(* PLC project Adressering.ecp, WAGO e!COCKPIT e!COCKPIT *)
(* stored: creationDateTime 2021-01-18T14:20:23.2110188, modificationDateTime 2021-01-18T11:51:27.6823754 *)

TYPE dtRomtype_1 : STRUCT
  RB601_V : BOOL;  (* Bevegelse *)
END_STRUCT;
END_TYPE

TYPE dtRomtype_11 : STRUCT
  RB601_V : BOOL;  (* Bevegelse *)
  RB601_HVAC : BOOL;  (* HVAC signal *)
END_STRUCT;
END_TYPE

TYPE dtRomtype_111 : STRUCT
  RB601_V : BOOL;  (* Bevegelse *)
  RB601_HVAC : BOOL;  (* HVAC signal *)
  RT601_CT : REAL;  (* Rom temperatur *)
  RT601_SP_D : REAL;  (* Temperatur SP dag/komfort *)
  RT601_SP_S : REAL;  (* Temperatur SP standby *)
  RT601_SP_N : REAL;  (* Temperatur SP nattsenk *)
  RT601_SP_F : REAL;  (* Temperatur SP frostsikring *)
  RT601_CS : REAL;  (* Aktivt temperatur SP *)
  OPM : REAL;  (* Rom modus *)
  OPM_CV : REAL;  (* Rom modus verdi *)
END_STRUCT;
END_TYPE

TYPE dtRomtype_1111 : STRUCT
  RB601_V : BOOL;  (* Bevegelse *)
  RB601_HVAC : BOOL;  (* HVAC signal *)
  RT601_CT : REAL;  (* Rom temperatur *)
  RT601_SP_D : REAL;  (* Temperatur SP dag/komfort *)
  RT601_SP_S : REAL;  (* Temperatur SP standby *)
  RT601_SP_N : REAL;  (* Temperatur SP nattsenk *)
  RT601_SP_F : REAL;  (* Temperatur SP frostsikring *)
  RT601_CS : REAL;  (* Aktivt temperatur SP *)
  OPM : REAL;  (* Rom modus *)
  OPM_CV : REAL;  (* Rom modus verdi *)
  RY601_CV : REAL;  (* Co2 Nivaa *)
  RY601_SP : REAL;  (* Co2 SP *)
  RY601_OP : REAL;  (* Co2 paadrag *)
END_STRUCT;
END_TYPE

TYPE dtRomtype_11101 : STRUCT
  RB601_V : BOOL;  (* Bevegelse *)
  RB601_HVAC : BOOL;  (* HVAC signal *)
  RT601_CT : REAL;  (* Rom temperatur *)
  RT601_SP_D : REAL;  (* Temperatur SP dag/komfort *)
  RT601_SP_S : REAL;  (* Temperatur SP standby *)
  RT601_SP_N : REAL;  (* Temperatur SP nattsenk *)
  RT601_SP_F : REAL;  (* Temperatur SP frostsikring *)
  RT601_CS : REAL;  (* Aktivt temperatur SP *)
  OPM : REAL;  (* Rom modus *)
  OPM_CV : REAL;  (* Rom modus verdi *)
  LH601_OP : REAL;  (* Varmepaadrag *)
  SB601_MAN : REAL;  (* Varmepaadrag force *)
END_STRUCT;
END_TYPE

TYPE dtRomtype_111011 : STRUCT
  RB601_V : BOOL;  (* Bevegelse *)
  RB601_HVAC : BOOL;  (* HVAC signal *)
  RT601_CT : REAL;  (* Rom temperatur *)
  RT601_SP_D : REAL;  (* Temperatur SP dag/komfort *)
  RT601_SP_S : REAL;  (* Temperatur SP standby *)
  RT601_SP_N : REAL;  (* Temperatur SP nattsenk *)
  RT601_SP_F : REAL;  (* Temperatur SP frostsikring *)
  RT601_CS : REAL;  (* Aktivt temperatur SP *)
  OPM : REAL;  (* Rom modus *)
  OPM_CV : REAL;  (* Rom modus verdi *)
  LH601_OP : REAL;  (* Varmepaadrag *)
  SB601_MAN : REAL;  (* Varmepaadrag force *)
  LH601_CMD : BOOL;  (* LH601_CMD *)
END_STRUCT;
END_TYPE

TYPE dtRomtype_1110111 : STRUCT
  RB601_V : BOOL;  (* Bevegelse *)
  RB601_HVAC : BOOL;  (* HVAC signal *)
  RT601_CT : REAL;  (* Rom temperatur *)
  RT601_SP_D : REAL;  (* Temperatur SP dag/komfort *)
  RT601_SP_S : REAL;  (* Temperatur SP standby *)
  RT601_SP_N : REAL;  (* Temperatur SP nattsenk *)
  RT601_SP_F : REAL;  (* Temperatur SP frostsikring *)
  RT601_CS : REAL;  (* Aktivt temperatur SP *)
  OPM : REAL;  (* Rom modus *)
  OPM_CV : REAL;  (* Rom modus verdi *)
  LH601_OP : REAL;  (* Varmepaadrag *)
  SB601_MAN : REAL;  (* Varmepaadrag force *)
  LH601_CMD : BOOL;  (* LH601_CMD *)
  LC601_OP : REAL;  (* LC601_OP *)
  LC601_MAN : REAL;  (* LC601 Force *)
END_STRUCT;
END_TYPE

TYPE dtRomtype_11111111 : STRUCT
  RB601_V : BOOL;  (* Bevegelse *)
  RB601_HVAC : BOOL;  (* HVAC signal *)
  RT601_CT : REAL;  (* Rom temperatur *)
  RT601_SP_D : REAL;  (* Temperatur SP dag/komfort *)
  RT601_SP_S : REAL;  (* Temperatur SP standby *)
  RT601_SP_N : REAL;  (* Temperatur SP nattsenk *)
  RT601_SP_F : REAL;  (* Temperatur SP frostsikring *)
  RT601_CS : REAL;  (* Aktivt temperatur SP *)
  OPM : REAL;  (* Rom modus *)
  OPM_CV : REAL;  (* Rom modus verdi *)
  RY601_CV : REAL;  (* Co2 Nivaa *)
  RY601_SP : REAL;  (* Co2 SP *)
  RY601_OP : REAL;  (* Co2 paadrag *)
  LH601_OP : REAL;  (* Varmepaadrag *)
  SB601_MAN : REAL;  (* Varmepaadrag force *)
  LH601_CMD : BOOL;  (* LH601_CMD *)
  LC601_OP : REAL;  (* LC601_OP *)
  LC601_MAN : REAL;  (* LC601 Force *)
  LC601_CMD : BOOL;  (* LC601_CMD *)
END_STRUCT;
END_TYPE

TYPE dtRomtype_111010111 : STRUCT
  RB601_V : BOOL;  (* Bevegelse *)
  RB601_HVAC : BOOL;  (* HVAC signal *)
  RT601_CT : REAL;  (* Rom temperatur *)
  RT601_SP_D : REAL;  (* Temperatur SP dag/komfort *)
  RT601_SP_S : REAL;  (* Temperatur SP standby *)
  RT601_SP_N : REAL;  (* Temperatur SP nattsenk *)
  RT601_SP_F : REAL;  (* Temperatur SP frostsikring *)
  RT601_CS : REAL;  (* Aktivt temperatur SP *)
  OPM : REAL;  (* Rom modus *)
  OPM_CV : REAL;  (* Rom modus verdi *)
  LH601_OP : REAL;  (* Varmepaadrag *)
  SB601_MAN : REAL;  (* Varmepaadrag force *)
  LC601_OP : REAL;  (* LC601_OP *)
  LC601_MAN : REAL;  (* LC601 Force *)
  LC601_CMD : BOOL;  (* LC601_CMD *)
  RT601_SP : REAL;  (* Temperatur SP feedback *)
END_STRUCT;
END_TYPE

TYPE dtRomtype_1111101011 : STRUCT
  RB601_V : BOOL;  (* Bevegelse *)
  RB601_HVAC : BOOL;  (* HVAC signal *)
  RT601_CT : REAL;  (* Rom temperatur *)
  RT601_SP_D : REAL;  (* Temperatur SP dag/komfort *)
  RT601_SP_S : REAL;  (* Temperatur SP standby *)
  RT601_SP_N : REAL;  (* Temperatur SP nattsenk *)
  RT601_SP_F : REAL;  (* Temperatur SP frostsikring *)
  RT601_CS : REAL;  (* Aktivt temperatur SP *)
  OPM : REAL;  (* Rom modus *)
  OPM_CV : REAL;  (* Rom modus verdi *)
  RY601_CV : REAL;  (* Co2 Nivaa *)
  RY601_SP : REAL;  (* Co2 SP *)
  RY601_OP : REAL;  (* Co2 paadrag *)
  LH601_OP : REAL;  (* Varmepaadrag *)
  SB601_MAN : REAL;  (* Varmepaadrag force *)
  LC601_OP : REAL;  (* LC601_OP *)
  LC601_MAN : REAL;  (* LC601 Force *)
  RT601_SP : REAL;  (* Temperatur SP feedback *)
  RT601_SP_FB : REAL;  (* Temperatur SP *)
  RT601_SP_IN : REAL;  (* Temperatur SP lokalt panel *)
END_STRUCT;
END_TYPE

TYPE dtRomtype_1111111111 : STRUCT
  RB601_V : BOOL;  (* Bevegelse *)
  RB601_HVAC : BOOL;  (* HVAC signal *)
  RT601_CT : REAL;  (* Rom temperatur *)
  RT601_SP_D : REAL;  (* Temperatur SP dag/komfort *)
  RT601_SP_S : REAL;  (* Temperatur SP standby *)
  RT601_SP_N : REAL;  (* Temperatur SP nattsenk *)
  RT601_SP_F : REAL;  (* Temperatur SP frostsikring *)
  RT601_CS : REAL;  (* Aktivt temperatur SP *)
  OPM : REAL;  (* Rom modus *)
  OPM_CV : REAL;  (* Rom modus verdi *)
  RY601_CV : REAL;  (* Co2 Nivaa *)
  RY601_SP : REAL;  (* Co2 SP *)
  RY601_OP : REAL;  (* Co2 paadrag *)
  LH601_OP : REAL;  (* Varmepaadrag *)
  SB601_MAN : REAL;  (* Varmepaadrag force *)
  LH601_CMD : BOOL;  (* LH601_CMD *)
  LC601_OP : REAL;  (* LC601_OP *)
  LC601_MAN : REAL;  (* LC601 Force *)
  LC601_CMD : BOOL;  (* LC601_CMD *)
  RT601_SP : REAL;  (* Temperatur SP feedback *)
  RT601_SP_FB : REAL;  (* Temperatur SP *)
  RT601_SP_IN : REAL;  (* Temperatur SP lokalt panel *)
END_STRUCT;
END_TYPE

{attribute 'qualified_only'}
VAR_GLOBAL  (* STLV80_563 *)
  STLV80_A_563_KNX_Card_1_Status : BOOL;  (* KNX kort 1 status *)
  STLV80_A_563_5A201 : dtRomtype_1;  (* rom1 *)
  STLV80_A_563_5A202 : dtRomtype_11;  (* rom1 *)
  STLV80_A_563_5A301 : dtRomtype_111;  (* rom1 *)
  STLV80_A_563_5A302 : dtRomtype_1111;  (* rom1 *)
  STLV80_A_563_5B201 : dtRomtype_11101;  (* rom1 *)
  STLV80_A_563_5B202 : dtRomtype_111011;  (* rom1 *)
  STLV80_A_563_5B301 : dtRomtype_1110111;  (* rom1 *)
  STLV80_A_563_5B302 : dtRomtype_11111111;  (* rom1 *)
  STLV80_A_563_5C201 : dtRomtype_111010111;  (* rom1 *)
  STLV80_A_563_5C202 : dtRomtype_1111101011;  (* rom1 *)
  STLV80_A_563_5C301 : dtRomtype_11111111;  (* rom1 *)
  STLV80_A_563_5C302 : dtRomtype_1111111111;  (* rom1 *)
  STLV80_A_563_5D201 : dtRomtype_1111111111;  (* rom1 *)
  STLV80_A_563_5D202 : dtRomtype_1111111111;  (* rom1 *)
  STLV80_A_563_5D301 : dtRomtype_1111111111;  (* rom1 *)
  STLV80_A_563_5D302 : dtRomtype_1111111111;  (* rom1 *)
END_VAR

PROGRAM PRG_563_KNX_1
  VAR
    i : INT := 0;  (* Felles *)
    Interval : OSCAT_BASIC.CLK_PRG;
    typDPT : typDPT;
    KNX_master_1 : WagoAppKNX.FbKNX_Master;  (* Master *)
    M1_001_5A201_RB601_V : fbDPT_Switch_pro;  (* 5A201 *)
    M1_002_5A202_RB601_V : fbDPT_Switch_pro;  (* 5A202 *)
    M1_003_5A202_RB601_HVAC : fbDPT_Switch_pro;  (* 5A202 *)
    M1_004_5A301_RB601_V : fbDPT_Switch_pro;  (* 5A301 *)
    M1_005_5A301_RB601_HVAC : fbDPT_Switch_pro;  (* 5A301 *)
    M1_006_5A301_RT601_CT : fbDPT_Value_Temp_pro;  (* 5A301 *)
    M1_007_5A302_RB601_V : fbDPT_Switch_pro;  (* 5A302 *)
    M1_008_5A302_RB601_HVAC : fbDPT_Switch_pro;  (* 5A302 *)
    M1_009_5A302_RT601_CT : fbDPT_Value_Temp_pro;  (* 5A302 *)
    M1_010_5A302_RY601_CV : fbDPT_Value_AirQuality_pro;  (* 5A302 *)
    M1_011_5B201_RB601_V : fbDPT_Switch_pro;  (* 5B201 *)
    M1_012_5B201_RB601_HVAC : fbDPT_Switch_pro;  (* 5B201 *)
    M1_013_5B201_RT601_CT : fbDPT_Value_Temp_pro;  (* 5B201 *)
    M1_014_5B201_LH601_OP : fbDPT_Scaling_pro;  (* 5B201 *)
    M1_015_5B202_RB601_V : fbDPT_Switch_pro;  (* 5B202 *)
    M1_016_5B202_RB601_HVAC : fbDPT_Switch_pro;  (* 5B202 *)
    M1_017_5B202_RT601_CT : fbDPT_Value_Temp_pro;  (* 5B202 *)
    M1_018_5B202_LH601_OP : fbDPT_Scaling_pro;  (* 5B202 *)
    M1_019_5B202_LH601_CMD : fbDPT_Switch_pro;  (* 5B202 *)
    M1_020_5B301_RB601_V : fbDPT_Switch_pro;  (* 5B301 *)
    M1_021_5B301_RB601_HVAC : fbDPT_Switch_pro;  (* 5B301 *)
    M1_022_5B301_RT601_CT : fbDPT_Value_Temp_pro;  (* 5B301 *)
    M1_023_5B301_LH601_OP : fbDPT_Scaling_pro;  (* 5B301 *)
    M1_024_5B301_LH601_CMD : fbDPT_Switch_pro;  (* 5B301 *)
    M1_025_5B301_LC601_OP : fbDPT_Scaling_pro;  (* 5B301 *)
    M1_026_5B302_RB601_V : fbDPT_Switch_pro;  (* 5B302 *)
    M1_027_5B302_RB601_HVAC : fbDPT_Switch_pro;  (* 5B302 *)
    M1_028_5B302_RT601_CT : fbDPT_Value_Temp_pro;  (* 5B302 *)
    M1_029_5B302_RY601_CV : fbDPT_Value_AirQuality_pro;  (* 5B302 *)
    M1_030_5B302_LH601_OP : fbDPT_Scaling_pro;  (* 5B302 *)
    M1_031_5B302_LH601_CMD : fbDPT_Switch_pro;  (* 5B302 *)
    M1_032_5B302_LC601_OP : fbDPT_Scaling_pro;  (* 5B302 *)
    M1_033_5B302_LC601_CMD : fbDPT_Switch_pro;  (* 5B302 *)
    M1_034_5C201_RB601_V : fbDPT_Switch_pro;  (* 5C201 *)
    M1_035_5C201_RB601_HVAC : fbDPT_Switch_pro;  (* 5C201 *)
    M1_036_5C201_RT601_CT : fbDPT_Value_Temp_pro;  (* 5C201 *)
    M1_037_5C201_LH601_OP : fbDPT_Scaling_pro;  (* 5C201 *)
    M1_038_5C201_LC601_OP : fbDPT_Scaling_pro;  (* 5C201 *)
    M1_039_5C201_LC601_CMD : fbDPT_Switch_pro;  (* 5C201 *)
    M1_040_5C201_RT601_SP : fbDPT_Value_Temp_pro;  (* 5C201 *)
    M1_041_5C202_RB601_V : fbDPT_Switch_pro;  (* 5C202 *)
    M1_042_5C202_RB601_HVAC : fbDPT_Switch_pro;  (* 5C202 *)
    M1_043_5C202_RT601_CT : fbDPT_Value_Temp_pro;  (* 5C202 *)
    M1_044_5C202_RY601_CV : fbDPT_Value_AirQuality_pro;  (* 5C202 *)
    M1_045_5C202_LH601_OP : fbDPT_Scaling_pro;  (* 5C202 *)
    M1_046_5C202_LC601_OP : fbDPT_Scaling_pro;  (* 5C202 *)
    M1_047_5C202_RT601_SP : fbDPT_Value_Temp_pro;  (* 5C202 *)
    M1_048_5C202_RT601_SP_FB : fbDPT_Value_Temp_pro;  (* 5C202 *)
    M1_049_5C301_RB601_V : fbDPT_Switch_pro;  (* 5C301 *)
    M1_050_5C301_RB601_HVAC : fbDPT_Switch_pro;  (* 5C301 *)
    M1_051_5C301_RT601_CT : fbDPT_Value_Temp_pro;  (* 5C301 *)
    M1_052_5C301_RY601_CV : fbDPT_Value_AirQuality_pro;  (* 5C301 *)
    M1_053_5C301_LH601_OP : fbDPT_Scaling_pro;  (* 5C301 *)
    M1_054_5C301_LH601_CMD : fbDPT_Switch_pro;  (* 5C301 *)
    M1_055_5C301_LC601_OP : fbDPT_Scaling_pro;  (* 5C301 *)
    M1_056_5C301_LC601_CMD : fbDPT_Switch_pro;  (* 5C301 *)
    M1_057_5C302_RB601_V : fbDPT_Switch_pro;  (* 5C302 *)
    M1_058_5C302_RB601_HVAC : fbDPT_Switch_pro;  (* 5C302 *)
    M1_059_5C302_RT601_CT : fbDPT_Value_Temp_pro;  (* 5C302 *)
    M1_060_5C302_RY601_CV : fbDPT_Value_AirQuality_pro;  (* 5C302 *)
    M1_061_5C302_LH601_OP : fbDPT_Scaling_pro;  (* 5C302 *)
    M1_062_5C302_LH601_CMD : fbDPT_Switch_pro;  (* 5C302 *)
    M1_063_5C302_LC601_OP : fbDPT_Scaling_pro;  (* 5C302 *)
    M1_064_5C302_LC601_CMD : fbDPT_Switch_pro;  (* 5C302 *)
    M1_065_5C302_RT601_SP : fbDPT_Value_Temp_pro;  (* 5C302 *)
    M1_066_5C302_RT601_SP_FB : fbDPT_Value_Temp_pro;  (* 5C302 *)
    M1_067_5D201_RB601_V : fbDPT_Switch_pro;  (* 5D201 *)
    M1_068_5D201_RB601_HVAC : fbDPT_Switch_pro;  (* 5D201 *)
    M1_069_5D201_RT601_CT : fbDPT_Value_Temp_pro;  (* 5D201 *)
    M1_070_5D201_RY601_CV : fbDPT_Value_AirQuality_pro;  (* 5D201 *)
    M1_071_5D201_LH601_OP : fbDPT_Scaling_pro;  (* 5D201 *)
    M1_072_5D201_LH601_CMD : fbDPT_Switch_pro;  (* 5D201 *)
    M1_073_5D201_LC601_OP : fbDPT_Scaling_pro;  (* 5D201 *)
    M1_074_5D201_LC601_CMD : fbDPT_Switch_pro;  (* 5D201 *)
    M1_075_5D201_RT601_SP : fbDPT_Value_Temp_pro;  (* 5D201 *)
    M1_076_5D201_RT601_SP_FB : fbDPT_Value_Temp_pro;  (* 5D201 *)
    M1_077_5D202_RB601_V : fbDPT_Switch_pro;  (* 5D202 *)
    M1_078_5D202_RB601_HVAC : fbDPT_Switch_pro;  (* 5D202 *)
    M1_079_5D202_RT601_CT : fbDPT_Value_Temp_pro;  (* 5D202 *)
    M1_080_5D202_RY601_CV : fbDPT_Value_AirQuality_pro;  (* 5D202 *)
    M1_081_5D202_LH601_OP : fbDPT_Scaling_pro;  (* 5D202 *)
    M1_082_5D202_LH601_CMD : fbDPT_Switch_pro;  (* 5D202 *)
    M1_083_5D202_LC601_OP : fbDPT_Scaling_pro;  (* 5D202 *)
    M1_084_5D202_LC601_CMD : fbDPT_Switch_pro;  (* 5D202 *)
    M1_085_5D202_RT601_SP : fbDPT_Value_Temp_pro;  (* 5D202 *)
    M1_086_5D202_RT601_SP_FB : fbDPT_Value_Temp_pro;  (* 5D202 *)
    M1_087_5D301_RB601_V : fbDPT_Switch_pro;  (* 5D301 *)
    M1_088_5D301_RB601_HVAC : fbDPT_Switch_pro;  (* 5D301 *)
    M1_089_5D301_RT601_CT : fbDPT_Value_Temp_pro;  (* 5D301 *)
    M1_090_5D301_RY601_CV : fbDPT_Value_AirQuality_pro;  (* 5D301 *)
    M1_091_5D301_LH601_OP : fbDPT_Scaling_pro;  (* 5D301 *)
    M1_092_5D301_LH601_CMD : fbDPT_Switch_pro;  (* 5D301 *)
    M1_093_5D301_LC601_OP : fbDPT_Scaling_pro;  (* 5D301 *)
    M1_094_5D301_LC601_CMD : fbDPT_Switch_pro;  (* 5D301 *)
    M1_095_5D301_RT601_SP : fbDPT_Value_Temp_pro;  (* 5D301 *)
    M1_096_5D301_RT601_SP_FB : fbDPT_Value_Temp_pro;  (* 5D301 *)
    M1_097_5D302_RB601_V : fbDPT_Switch_pro;  (* 5D302 *)
    M1_098_5D302_RB601_HVAC : fbDPT_Switch_pro;  (* 5D302 *)
    M1_099_5D302_RT601_CT : fbDPT_Value_Temp_pro;  (* 5D302 *)
    M1_100_5D302_RY601_CV : fbDPT_Value_AirQuality_pro;  (* 5D302 *)
    M1_101_5D302_LH601_OP : fbDPT_Scaling_pro;  (* 5D302 *)
    M1_102_5D302_LH601_CMD : fbDPT_Switch_pro;  (* 5D302 *)
    M1_103_5D302_LC601_OP : fbDPT_Scaling_pro;  (* 5D302 *)
    M1_104_5D302_LC601_CMD : fbDPT_Switch_pro;  (* 5D302 *)
    M1_105_5D302_RT601_SP : fbDPT_Value_Temp_pro;  (* 5D302 *)
    M1_106_5D302_RT601_SP_FB : fbDPT_Value_Temp_pro;  (* 5D302 *)
  END_VAR
  VAR  (* added by the conversion: wires and edge detectors of the diagram *)
    _ADD9_OUT : INT;
    _GT15_OUT : BOOL;
    _MOVE19_ENO : BOOL;
    _MOVE19_OUT : INT;
  END_VAR

(* CFC diagram, written out as Structured Text *)
(* KNX Sending interval *)
(* KNX Master *)
Interval(PT := t#2M);
_ADD9_OUT := BOOL_TO_INT(Interval.Q) + i;
i := _ADD9_OUT;
_GT15_OUT := i > 39;
_MOVE19_OUT := MOVE(EN := _GT15_OUT, IN := 0, ENO => _MOVE19_ENO);
IF _MOVE19_ENO THEN i := _MOVE19_OUT; END_IF;
KNX_master_1(I_Port := IoConfig_Globals.KNX_EIB_TP1_Interface, bPortKNX := 1);
STLV80_563.STLV80_A_563_KNX_Card_1_Status := KNX_master_1.sStatus = 'OK';
(* Rom 5A201 *)
(* RB601_V *)
M1_001_5A201_RB601_V(bPortKNX := 1, dwIndex_DPT := 1, typDPT := typDPT);
STLV80_563.STLV80_A_563_5A201.RB601_V := M1_001_5A201_RB601_V.xSwitch_OUT;
(* Rom 5A202 *)
(* RB601_V *)
(* RB601_HVAC *)
M1_002_5A202_RB601_V(bPortKNX := 1, dwIndex_DPT := 2, typDPT := typDPT);
STLV80_563.STLV80_A_563_5A202.RB601_V := M1_002_5A202_RB601_V.xSwitch_OUT;
M1_003_5A202_RB601_HVAC(bPortKNX := 1, dwIndex_DPT := 3, typDPT := typDPT);
STLV80_563.STLV80_A_563_5A202.RB601_HVAC := M1_003_5A202_RB601_HVAC.xSwitch_OUT;
(* Rom 5A301 *)
(* RB601_V *)
(* RB601_HVAC *)
M1_004_5A301_RB601_V(bPortKNX := 1, dwIndex_DPT := 4, typDPT := typDPT);
STLV80_563.STLV80_A_563_5A301.RB601_V := M1_004_5A301_RB601_V.xSwitch_OUT;
M1_005_5A301_RB601_HVAC(bPortKNX := 1, dwIndex_DPT := 5, typDPT := typDPT);
STLV80_563.STLV80_A_563_5A301.RB601_HVAC := M1_005_5A301_RB601_HVAC.xSwitch_OUT;
(* RT601_CT *)
M1_006_5A301_RT601_CT(bPortKNX := 1, dwIndex_DPT := 6, typDPT := typDPT);
STLV80_563.STLV80_A_563_5A301.RT601_CT := M1_006_5A301_RT601_CT.rValue_OUT;
(* Rom 5A302 *)
(* RB601_V *)
(* RB601_HVAC *)
M1_007_5A302_RB601_V(bPortKNX := 1, dwIndex_DPT := 7, typDPT := typDPT);
STLV80_563.STLV80_A_563_5A302.RB601_V := M1_007_5A302_RB601_V.xSwitch_OUT;
M1_008_5A302_RB601_HVAC(bPortKNX := 1, dwIndex_DPT := 8, typDPT := typDPT);
STLV80_563.STLV80_A_563_5A302.RB601_HVAC := M1_008_5A302_RB601_HVAC.xSwitch_OUT;
(* RT601_CT *)
(* RY601_CV *)
M1_009_5A302_RT601_CT(bPortKNX := 1, dwIndex_DPT := 9, typDPT := typDPT);
STLV80_563.STLV80_A_563_5A302.RT601_CT := M1_009_5A302_RT601_CT.rValue_OUT;
M1_010_5A302_RY601_CV(bPortKNX := 1, dwIndex_DPT := 10, typDPT := typDPT);
STLV80_563.STLV80_A_563_5A302.RY601_CV := M1_010_5A302_RY601_CV.rValue_OUT;
(* Rom 5B201 *)
(* RB601_V *)
(* RB601_HVAC *)
M1_011_5B201_RB601_V(bPortKNX := 1, dwIndex_DPT := 11, typDPT := typDPT);
STLV80_563.STLV80_A_563_5B201.RB601_V := M1_011_5B201_RB601_V.xSwitch_OUT;
M1_012_5B201_RB601_HVAC(bPortKNX := 1, dwIndex_DPT := 12, typDPT := typDPT);
STLV80_563.STLV80_A_563_5B201.RB601_HVAC := M1_012_5B201_RB601_HVAC.xSwitch_OUT;
(* RT601_CT *)
(* LH601_OP *)
M1_013_5B201_RT601_CT(bPortKNX := 1, dwIndex_DPT := 13, typDPT := typDPT);
STLV80_563.STLV80_A_563_5B201.RT601_CT := M1_013_5B201_RT601_CT.rValue_OUT;
M1_014_5B201_LH601_OP(bPortKNX := 1, dwIndex_DPT := 14, rValue_IN := STLV80_563.STLV80_A_563_5B201.LH601_OP, xUpdate_KNX := i = 0, typDPT := typDPT);
(* Rom 5B202 *)
(* RB601_V *)
(* RB601_HVAC *)
M1_015_5B202_RB601_V(bPortKNX := 1, dwIndex_DPT := 15, typDPT := typDPT);
STLV80_563.STLV80_A_563_5B202.RB601_V := M1_015_5B202_RB601_V.xSwitch_OUT;
M1_016_5B202_RB601_HVAC(bPortKNX := 1, dwIndex_DPT := 16, typDPT := typDPT);
STLV80_563.STLV80_A_563_5B202.RB601_HVAC := M1_016_5B202_RB601_HVAC.xSwitch_OUT;
(* RT601_CT *)
(* LH601_OP *)
M1_017_5B202_RT601_CT(bPortKNX := 1, dwIndex_DPT := 17, typDPT := typDPT);
STLV80_563.STLV80_A_563_5B202.RT601_CT := M1_017_5B202_RT601_CT.rValue_OUT;
M1_018_5B202_LH601_OP(bPortKNX := 1, dwIndex_DPT := 18, rValue_IN := STLV80_563.STLV80_A_563_5B202.LH601_OP, xUpdate_KNX := i = 1, typDPT := typDPT);
(* LH601_CMD *)
M1_019_5B202_LH601_CMD(bPortKNX := 1, dwIndex_DPT := 19, xSwitch_IN := STLV80_563.STLV80_A_563_5B202.LH601_CMD, xUpdate_KNX := i = 2, typDPT := typDPT);
(* Rom 5B301 *)
(* RB601_V *)
(* RB601_HVAC *)
M1_020_5B301_RB601_V(bPortKNX := 1, dwIndex_DPT := 20, typDPT := typDPT);
STLV80_563.STLV80_A_563_5B301.RB601_V := M1_020_5B301_RB601_V.xSwitch_OUT;
M1_021_5B301_RB601_HVAC(bPortKNX := 1, dwIndex_DPT := 21, typDPT := typDPT);
STLV80_563.STLV80_A_563_5B301.RB601_HVAC := M1_021_5B301_RB601_HVAC.xSwitch_OUT;
(* RT601_CT *)
(* LH601_OP *)
M1_022_5B301_RT601_CT(bPortKNX := 1, dwIndex_DPT := 22, typDPT := typDPT);
STLV80_563.STLV80_A_563_5B301.RT601_CT := M1_022_5B301_RT601_CT.rValue_OUT;
M1_023_5B301_LH601_OP(bPortKNX := 1, dwIndex_DPT := 23, rValue_IN := STLV80_563.STLV80_A_563_5B301.LH601_OP, xUpdate_KNX := i = 3, typDPT := typDPT);
(* LH601_CMD *)
(* LC601_OP *)
M1_024_5B301_LH601_CMD(bPortKNX := 1, dwIndex_DPT := 24, xSwitch_IN := STLV80_563.STLV80_A_563_5B301.LH601_CMD, xUpdate_KNX := i = 4, typDPT := typDPT);
M1_025_5B301_LC601_OP(bPortKNX := 1, dwIndex_DPT := 25, rValue_IN := STLV80_563.STLV80_A_563_5B301.LC601_OP, xUpdate_KNX := i = 5, typDPT := typDPT);
(* Rom 5B302 *)
(* RB601_V *)
(* RB601_HVAC *)
M1_026_5B302_RB601_V(bPortKNX := 1, dwIndex_DPT := 26, typDPT := typDPT);
STLV80_563.STLV80_A_563_5B302.RB601_V := M1_026_5B302_RB601_V.xSwitch_OUT;
M1_027_5B302_RB601_HVAC(bPortKNX := 1, dwIndex_DPT := 27, typDPT := typDPT);
STLV80_563.STLV80_A_563_5B302.RB601_HVAC := M1_027_5B302_RB601_HVAC.xSwitch_OUT;
(* RT601_CT *)
(* RY601_CV *)
M1_028_5B302_RT601_CT(bPortKNX := 1, dwIndex_DPT := 28, typDPT := typDPT);
STLV80_563.STLV80_A_563_5B302.RT601_CT := M1_028_5B302_RT601_CT.rValue_OUT;
M1_029_5B302_RY601_CV(bPortKNX := 1, dwIndex_DPT := 29, typDPT := typDPT);
STLV80_563.STLV80_A_563_5B302.RY601_CV := M1_029_5B302_RY601_CV.rValue_OUT;
(* LH601_OP *)
(* LH601_CMD *)
M1_030_5B302_LH601_OP(bPortKNX := 1, dwIndex_DPT := 30, rValue_IN := STLV80_563.STLV80_A_563_5B302.LH601_OP, xUpdate_KNX := i = 6, typDPT := typDPT);
M1_031_5B302_LH601_CMD(bPortKNX := 1, dwIndex_DPT := 31, xSwitch_IN := STLV80_563.STLV80_A_563_5B302.LH601_CMD, xUpdate_KNX := i = 7, typDPT := typDPT);
(* LC601_OP *)
(* LC601_CMD *)
M1_032_5B302_LC601_OP(bPortKNX := 1, dwIndex_DPT := 32, rValue_IN := STLV80_563.STLV80_A_563_5B302.LC601_OP, xUpdate_KNX := i = 8, typDPT := typDPT);
M1_033_5B302_LC601_CMD(bPortKNX := 1, dwIndex_DPT := 33, xSwitch_IN := STLV80_563.STLV80_A_563_5B302.LC601_CMD, xUpdate_KNX := i = 9, typDPT := typDPT);
(* Rom 5C201 *)
(* RB601_V *)
(* RB601_HVAC *)
M1_034_5C201_RB601_V(bPortKNX := 1, dwIndex_DPT := 34, typDPT := typDPT);
STLV80_563.STLV80_A_563_5C201.RB601_V := M1_034_5C201_RB601_V.xSwitch_OUT;
M1_035_5C201_RB601_HVAC(bPortKNX := 1, dwIndex_DPT := 35, typDPT := typDPT);
STLV80_563.STLV80_A_563_5C201.RB601_HVAC := M1_035_5C201_RB601_HVAC.xSwitch_OUT;
(* RT601_CT *)
(* LH601_OP *)
M1_036_5C201_RT601_CT(bPortKNX := 1, dwIndex_DPT := 36, typDPT := typDPT);
STLV80_563.STLV80_A_563_5C201.RT601_CT := M1_036_5C201_RT601_CT.rValue_OUT;
M1_037_5C201_LH601_OP(bPortKNX := 1, dwIndex_DPT := 37, rValue_IN := STLV80_563.STLV80_A_563_5C201.LH601_OP, xUpdate_KNX := i = 10, typDPT := typDPT);
(* LC601_OP *)
(* LC601_CMD *)
M1_038_5C201_LC601_OP(bPortKNX := 1, dwIndex_DPT := 38, rValue_IN := STLV80_563.STLV80_A_563_5C201.LC601_OP, xUpdate_KNX := i = 11, typDPT := typDPT);
M1_039_5C201_LC601_CMD(bPortKNX := 1, dwIndex_DPT := 39, xSwitch_IN := STLV80_563.STLV80_A_563_5C201.LC601_CMD, xUpdate_KNX := i = 12, typDPT := typDPT);
(* RT601_SP *)
M1_040_5C201_RT601_SP(bPortKNX := 1, dwIndex_DPT := 40, rValue_IN := STLV80_563.STLV80_A_563_5C201.RT601_SP_D, xUpdate_KNX := NOT STLV80_563.STLV80_A_563_5C201.RB601_HVAC, typDPT := typDPT);
(* Rom 5C202 *)
(* RB601_V *)
(* RB601_HVAC *)
M1_041_5C202_RB601_V(bPortKNX := 1, dwIndex_DPT := 41, typDPT := typDPT);
STLV80_563.STLV80_A_563_5C202.RB601_V := M1_041_5C202_RB601_V.xSwitch_OUT;
M1_042_5C202_RB601_HVAC(bPortKNX := 1, dwIndex_DPT := 42, typDPT := typDPT);
STLV80_563.STLV80_A_563_5C202.RB601_HVAC := M1_042_5C202_RB601_HVAC.xSwitch_OUT;
(* RT601_CT *)
(* RY601_CV *)
M1_043_5C202_RT601_CT(bPortKNX := 1, dwIndex_DPT := 43, typDPT := typDPT);
STLV80_563.STLV80_A_563_5C202.RT601_CT := M1_043_5C202_RT601_CT.rValue_OUT;
M1_044_5C202_RY601_CV(bPortKNX := 1, dwIndex_DPT := 44, typDPT := typDPT);
STLV80_563.STLV80_A_563_5C202.RY601_CV := M1_044_5C202_RY601_CV.rValue_OUT;
(* LH601_OP *)
(* LC601_OP *)
M1_045_5C202_LH601_OP(bPortKNX := 1, dwIndex_DPT := 45, rValue_IN := STLV80_563.STLV80_A_563_5C202.LH601_OP, xUpdate_KNX := i = 13, typDPT := typDPT);
M1_046_5C202_LC601_OP(bPortKNX := 1, dwIndex_DPT := 46, rValue_IN := STLV80_563.STLV80_A_563_5C202.LC601_OP, xUpdate_KNX := i = 14, typDPT := typDPT);
(* RT601_SP *)
(* RT601_SP Feedback *)
M1_047_5C202_RT601_SP(bPortKNX := 1, dwIndex_DPT := 47, rValue_IN := STLV80_563.STLV80_A_563_5C202.RT601_SP_D, xUpdate_KNX := NOT STLV80_563.STLV80_A_563_5C202.RB601_HVAC, typDPT := typDPT);
M1_048_5C202_RT601_SP_FB(bPortKNX := 1, dwIndex_DPT := 48, typDPT := typDPT);
STLV80_563.STLV80_A_563_5C202.RT601_SP_IN := M1_048_5C202_RT601_SP_FB.rValue_OUT;
(* Rom 5C301 *)
(* RB601_V *)
(* RB601_HVAC *)
M1_049_5C301_RB601_V(bPortKNX := 1, dwIndex_DPT := 49, typDPT := typDPT);
STLV80_563.STLV80_A_563_5C301.RB601_V := M1_049_5C301_RB601_V.xSwitch_OUT;
M1_050_5C301_RB601_HVAC(bPortKNX := 1, dwIndex_DPT := 50, typDPT := typDPT);
STLV80_563.STLV80_A_563_5C301.RB601_HVAC := M1_050_5C301_RB601_HVAC.xSwitch_OUT;
(* RT601_CT *)
(* RY601_CV *)
M1_051_5C301_RT601_CT(bPortKNX := 1, dwIndex_DPT := 51, typDPT := typDPT);
STLV80_563.STLV80_A_563_5C301.RT601_CT := M1_051_5C301_RT601_CT.rValue_OUT;
M1_052_5C301_RY601_CV(bPortKNX := 1, dwIndex_DPT := 52, typDPT := typDPT);
STLV80_563.STLV80_A_563_5C301.RY601_CV := M1_052_5C301_RY601_CV.rValue_OUT;
(* LH601_OP *)
(* LH601_CMD *)
M1_053_5C301_LH601_OP(bPortKNX := 1, dwIndex_DPT := 53, rValue_IN := STLV80_563.STLV80_A_563_5C301.LH601_OP, xUpdate_KNX := i = 15, typDPT := typDPT);
M1_054_5C301_LH601_CMD(bPortKNX := 1, dwIndex_DPT := 54, xSwitch_IN := STLV80_563.STLV80_A_563_5C301.LH601_CMD, xUpdate_KNX := i = 16, typDPT := typDPT);
(* LC601_OP *)
(* LC601_CMD *)
M1_055_5C301_LC601_OP(bPortKNX := 1, dwIndex_DPT := 55, rValue_IN := STLV80_563.STLV80_A_563_5C301.LC601_OP, xUpdate_KNX := i = 17, typDPT := typDPT);
M1_056_5C301_LC601_CMD(bPortKNX := 1, dwIndex_DPT := 56, xSwitch_IN := STLV80_563.STLV80_A_563_5C301.LC601_CMD, xUpdate_KNX := i = 18, typDPT := typDPT);
(* Rom 5C302 *)
(* RB601_V *)
(* RB601_HVAC *)
M1_057_5C302_RB601_V(bPortKNX := 1, dwIndex_DPT := 57, typDPT := typDPT);
STLV80_563.STLV80_A_563_5C302.RB601_V := M1_057_5C302_RB601_V.xSwitch_OUT;
M1_058_5C302_RB601_HVAC(bPortKNX := 1, dwIndex_DPT := 58, typDPT := typDPT);
STLV80_563.STLV80_A_563_5C302.RB601_HVAC := M1_058_5C302_RB601_HVAC.xSwitch_OUT;
(* RT601_CT *)
(* RY601_CV *)
M1_059_5C302_RT601_CT(bPortKNX := 1, dwIndex_DPT := 59, typDPT := typDPT);
STLV80_563.STLV80_A_563_5C302.RT601_CT := M1_059_5C302_RT601_CT.rValue_OUT;
M1_060_5C302_RY601_CV(bPortKNX := 1, dwIndex_DPT := 60, typDPT := typDPT);
STLV80_563.STLV80_A_563_5C302.RY601_CV := M1_060_5C302_RY601_CV.rValue_OUT;
(* LH601_OP *)
(* LH601_CMD *)
M1_061_5C302_LH601_OP(bPortKNX := 1, dwIndex_DPT := 61, rValue_IN := STLV80_563.STLV80_A_563_5C302.LH601_OP, xUpdate_KNX := i = 19, typDPT := typDPT);
M1_062_5C302_LH601_CMD(bPortKNX := 1, dwIndex_DPT := 62, xSwitch_IN := STLV80_563.STLV80_A_563_5C302.LH601_CMD, xUpdate_KNX := i = 20, typDPT := typDPT);
(* LC601_OP *)
(* LC601_CMD *)
M1_063_5C302_LC601_OP(bPortKNX := 1, dwIndex_DPT := 63, rValue_IN := STLV80_563.STLV80_A_563_5C302.LC601_OP, xUpdate_KNX := i = 21, typDPT := typDPT);
M1_064_5C302_LC601_CMD(bPortKNX := 1, dwIndex_DPT := 64, xSwitch_IN := STLV80_563.STLV80_A_563_5C302.LC601_CMD, xUpdate_KNX := i = 22, typDPT := typDPT);
(* RT601_SP *)
(* RT601_SP Feedback *)
M1_065_5C302_RT601_SP(bPortKNX := 1, dwIndex_DPT := 65, rValue_IN := STLV80_563.STLV80_A_563_5C302.RT601_SP_D, xUpdate_KNX := NOT STLV80_563.STLV80_A_563_5C302.RB601_HVAC, typDPT := typDPT);
M1_066_5C302_RT601_SP_FB(bPortKNX := 1, dwIndex_DPT := 66, typDPT := typDPT);
STLV80_563.STLV80_A_563_5C302.RT601_SP_IN := M1_066_5C302_RT601_SP_FB.rValue_OUT;
(* Rom 5D201 *)
(* RB601_V *)
(* RB601_HVAC *)
M1_067_5D201_RB601_V(bPortKNX := 1, dwIndex_DPT := 67, typDPT := typDPT);
STLV80_563.STLV80_A_563_5D201.RB601_V := M1_067_5D201_RB601_V.xSwitch_OUT;
M1_068_5D201_RB601_HVAC(bPortKNX := 1, dwIndex_DPT := 68, typDPT := typDPT);
STLV80_563.STLV80_A_563_5D201.RB601_HVAC := M1_068_5D201_RB601_HVAC.xSwitch_OUT;
(* RT601_CT *)
(* RY601_CV *)
M1_069_5D201_RT601_CT(bPortKNX := 1, dwIndex_DPT := 69, typDPT := typDPT);
STLV80_563.STLV80_A_563_5D201.RT601_CT := M1_069_5D201_RT601_CT.rValue_OUT;
M1_070_5D201_RY601_CV(bPortKNX := 1, dwIndex_DPT := 70, typDPT := typDPT);
STLV80_563.STLV80_A_563_5D201.RY601_CV := M1_070_5D201_RY601_CV.rValue_OUT;
(* LH601_OP *)
(* LH601_CMD *)
M1_071_5D201_LH601_OP(bPortKNX := 1, dwIndex_DPT := 71, rValue_IN := STLV80_563.STLV80_A_563_5D201.LH601_OP, xUpdate_KNX := i = 23, typDPT := typDPT);
M1_072_5D201_LH601_CMD(bPortKNX := 1, dwIndex_DPT := 72, xSwitch_IN := STLV80_563.STLV80_A_563_5D201.LH601_CMD, xUpdate_KNX := i = 24, typDPT := typDPT);
(* LC601_OP *)
(* LC601_CMD *)
M1_073_5D201_LC601_OP(bPortKNX := 1, dwIndex_DPT := 73, rValue_IN := STLV80_563.STLV80_A_563_5D201.LC601_OP, xUpdate_KNX := i = 25, typDPT := typDPT);
M1_074_5D201_LC601_CMD(bPortKNX := 1, dwIndex_DPT := 74, xSwitch_IN := STLV80_563.STLV80_A_563_5D201.LC601_CMD, xUpdate_KNX := i = 26, typDPT := typDPT);
(* RT601_SP *)
(* RT601_SP Feedback *)
M1_075_5D201_RT601_SP(bPortKNX := 1, dwIndex_DPT := 75, rValue_IN := STLV80_563.STLV80_A_563_5D201.RT601_SP_D, xUpdate_KNX := NOT STLV80_563.STLV80_A_563_5D201.RB601_HVAC, typDPT := typDPT);
M1_076_5D201_RT601_SP_FB(bPortKNX := 1, dwIndex_DPT := 76, typDPT := typDPT);
STLV80_563.STLV80_A_563_5D201.RT601_SP_IN := M1_076_5D201_RT601_SP_FB.rValue_OUT;
(* Rom 5D202 *)
(* RB601_V *)
(* RB601_HVAC *)
M1_077_5D202_RB601_V(bPortKNX := 1, dwIndex_DPT := 77, typDPT := typDPT);
STLV80_563.STLV80_A_563_5D202.RB601_V := M1_077_5D202_RB601_V.xSwitch_OUT;
M1_078_5D202_RB601_HVAC(bPortKNX := 1, dwIndex_DPT := 78, typDPT := typDPT);
STLV80_563.STLV80_A_563_5D202.RB601_HVAC := M1_078_5D202_RB601_HVAC.xSwitch_OUT;
(* RT601_CT *)
(* RY601_CV *)
M1_079_5D202_RT601_CT(bPortKNX := 1, dwIndex_DPT := 79, typDPT := typDPT);
STLV80_563.STLV80_A_563_5D202.RT601_CT := M1_079_5D202_RT601_CT.rValue_OUT;
M1_080_5D202_RY601_CV(bPortKNX := 1, dwIndex_DPT := 80, typDPT := typDPT);
STLV80_563.STLV80_A_563_5D202.RY601_CV := M1_080_5D202_RY601_CV.rValue_OUT;
(* LH601_OP *)
(* LH601_CMD *)
M1_081_5D202_LH601_OP(bPortKNX := 1, dwIndex_DPT := 81, rValue_IN := STLV80_563.STLV80_A_563_5D202.LH601_OP, xUpdate_KNX := i = 27, typDPT := typDPT);
M1_082_5D202_LH601_CMD(bPortKNX := 1, dwIndex_DPT := 82, xSwitch_IN := STLV80_563.STLV80_A_563_5D202.LH601_CMD, xUpdate_KNX := i = 28, typDPT := typDPT);
(* LC601_OP *)
(* LC601_CMD *)
M1_083_5D202_LC601_OP(bPortKNX := 1, dwIndex_DPT := 83, rValue_IN := STLV80_563.STLV80_A_563_5D202.LC601_OP, xUpdate_KNX := i = 29, typDPT := typDPT);
M1_084_5D202_LC601_CMD(bPortKNX := 1, dwIndex_DPT := 84, xSwitch_IN := STLV80_563.STLV80_A_563_5D202.LC601_CMD, xUpdate_KNX := i = 30, typDPT := typDPT);
(* RT601_SP *)
(* RT601_SP Feedback *)
M1_085_5D202_RT601_SP(bPortKNX := 1, dwIndex_DPT := 85, rValue_IN := STLV80_563.STLV80_A_563_5D202.RT601_SP_D, xUpdate_KNX := NOT STLV80_563.STLV80_A_563_5D202.RB601_HVAC, typDPT := typDPT);
M1_086_5D202_RT601_SP_FB(bPortKNX := 1, dwIndex_DPT := 86, typDPT := typDPT);
STLV80_563.STLV80_A_563_5D202.RT601_SP_IN := M1_086_5D202_RT601_SP_FB.rValue_OUT;
(* Rom 5D301 *)
(* RB601_V *)
(* RB601_HVAC *)
M1_087_5D301_RB601_V(bPortKNX := 1, dwIndex_DPT := 87, typDPT := typDPT);
STLV80_563.STLV80_A_563_5D301.RB601_V := M1_087_5D301_RB601_V.xSwitch_OUT;
M1_088_5D301_RB601_HVAC(bPortKNX := 1, dwIndex_DPT := 88, typDPT := typDPT);
STLV80_563.STLV80_A_563_5D301.RB601_HVAC := M1_088_5D301_RB601_HVAC.xSwitch_OUT;
(* RT601_CT *)
(* RY601_CV *)
M1_089_5D301_RT601_CT(bPortKNX := 1, dwIndex_DPT := 89, typDPT := typDPT);
STLV80_563.STLV80_A_563_5D301.RT601_CT := M1_089_5D301_RT601_CT.rValue_OUT;
M1_090_5D301_RY601_CV(bPortKNX := 1, dwIndex_DPT := 90, typDPT := typDPT);
STLV80_563.STLV80_A_563_5D301.RY601_CV := M1_090_5D301_RY601_CV.rValue_OUT;
(* LH601_OP *)
(* LH601_CMD *)
M1_091_5D301_LH601_OP(bPortKNX := 1, dwIndex_DPT := 91, rValue_IN := STLV80_563.STLV80_A_563_5D301.LH601_OP, xUpdate_KNX := i = 31, typDPT := typDPT);
M1_092_5D301_LH601_CMD(bPortKNX := 1, dwIndex_DPT := 92, xSwitch_IN := STLV80_563.STLV80_A_563_5D301.LH601_CMD, xUpdate_KNX := i = 32, typDPT := typDPT);
(* LC601_OP *)
(* LC601_CMD *)
M1_093_5D301_LC601_OP(bPortKNX := 1, dwIndex_DPT := 93, rValue_IN := STLV80_563.STLV80_A_563_5D301.LC601_OP, xUpdate_KNX := i = 33, typDPT := typDPT);
M1_094_5D301_LC601_CMD(bPortKNX := 1, dwIndex_DPT := 94, xSwitch_IN := STLV80_563.STLV80_A_563_5D301.LC601_CMD, xUpdate_KNX := i = 34, typDPT := typDPT);
(* RT601_SP *)
(* RT601_SP Feedback *)
M1_095_5D301_RT601_SP(bPortKNX := 1, dwIndex_DPT := 95, rValue_IN := STLV80_563.STLV80_A_563_5D301.RT601_SP_D, xUpdate_KNX := NOT STLV80_563.STLV80_A_563_5D301.RB601_HVAC, typDPT := typDPT);
M1_096_5D301_RT601_SP_FB(bPortKNX := 1, dwIndex_DPT := 96, typDPT := typDPT);
STLV80_563.STLV80_A_563_5D301.RT601_SP_IN := M1_096_5D301_RT601_SP_FB.rValue_OUT;
(* Rom 5D302 *)
(* RB601_V *)
(* RB601_HVAC *)
M1_097_5D302_RB601_V(bPortKNX := 1, dwIndex_DPT := 97, typDPT := typDPT);
STLV80_563.STLV80_A_563_5D302.RB601_V := M1_097_5D302_RB601_V.xSwitch_OUT;
M1_098_5D302_RB601_HVAC(bPortKNX := 1, dwIndex_DPT := 98, typDPT := typDPT);
STLV80_563.STLV80_A_563_5D302.RB601_HVAC := M1_098_5D302_RB601_HVAC.xSwitch_OUT;
(* RT601_CT *)
(* RY601_CV *)
M1_099_5D302_RT601_CT(bPortKNX := 1, dwIndex_DPT := 99, typDPT := typDPT);
STLV80_563.STLV80_A_563_5D302.RT601_CT := M1_099_5D302_RT601_CT.rValue_OUT;
M1_100_5D302_RY601_CV(bPortKNX := 1, dwIndex_DPT := 100, typDPT := typDPT);
STLV80_563.STLV80_A_563_5D302.RY601_CV := M1_100_5D302_RY601_CV.rValue_OUT;
(* LH601_OP *)
(* LH601_CMD *)
M1_101_5D302_LH601_OP(bPortKNX := 1, dwIndex_DPT := 101, rValue_IN := STLV80_563.STLV80_A_563_5D302.LH601_OP, xUpdate_KNX := i = 35, typDPT := typDPT);
M1_102_5D302_LH601_CMD(bPortKNX := 1, dwIndex_DPT := 102, xSwitch_IN := STLV80_563.STLV80_A_563_5D302.LH601_CMD, xUpdate_KNX := i = 36, typDPT := typDPT);
(* LC601_OP *)
(* LC601_CMD *)
M1_103_5D302_LC601_OP(bPortKNX := 1, dwIndex_DPT := 103, rValue_IN := STLV80_563.STLV80_A_563_5D302.LC601_OP, xUpdate_KNX := i = 37, typDPT := typDPT);
M1_104_5D302_LC601_CMD(bPortKNX := 1, dwIndex_DPT := 104, xSwitch_IN := STLV80_563.STLV80_A_563_5D302.LC601_CMD, xUpdate_KNX := i = 38, typDPT := typDPT);
(* RT601_SP *)
(* RT601_SP Feedback *)
M1_105_5D302_RT601_SP(bPortKNX := 1, dwIndex_DPT := 105, rValue_IN := STLV80_563.STLV80_A_563_5D302.RT601_SP_D, xUpdate_KNX := NOT STLV80_563.STLV80_A_563_5D302.RB601_HVAC, typDPT := typDPT);
M1_106_5D302_RT601_SP_FB(bPortKNX := 1, dwIndex_DPT := 106, typDPT := typDPT);
STLV80_563.STLV80_A_563_5D302.RT601_SP_IN := M1_106_5D302_RT601_SP_FB.rValue_OUT;
END_PROGRAM
